# B&R Automation Studio project prak2
Automation Studio 4.5.2.102

## Configuration Config1

### Task classes (Cpu.sw)
```
Cyclic#4:
  Program <- Program.prg
DataObjects: Acp10sys
NcDataObjects: acp10etxen <- acp10etxen.dob
VcDataObjects: LED <- LED.dob
Binaries: udbdef, TCData, vcfntttf, vcpdsw, vcpfmtcx, arial, vcmgr, vccovl, vcdsint, vcpdpp30, vcshared, LED02, LED03, vcpfpp30, LED01, vcalarm, vccbtn, vcptelo, vcgclass, vcdsloc, arialbd, vcrt, vctcal, vcbclass, vcfile, Role, ashwd, ashwac, asfw, iomap, sysconf, User, arconfig, Acp10map, acp10cfg
Libraries: Acp10man, Acp10par, NcGlobal, Acp10sdc, AsBrStr, powerlnk, astime, fileio, runtime, dataobj, vcresman
```

### Hardware
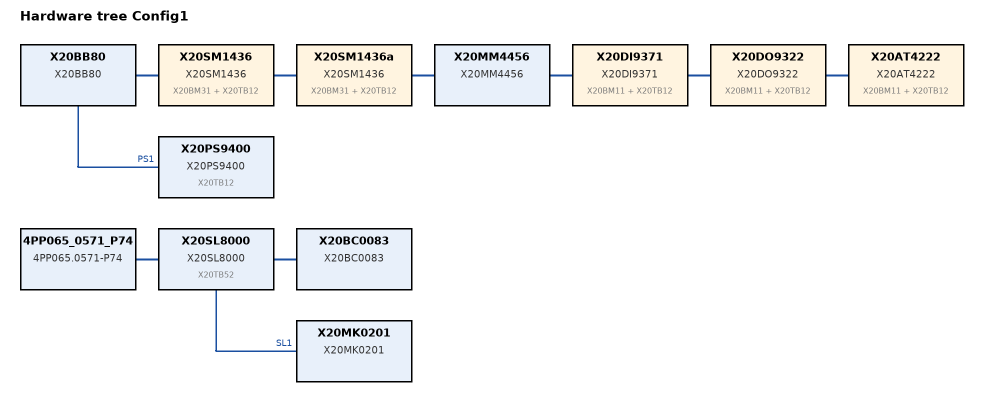
```
4PP065_0571_P74 : 4PP065.0571-P74 v1.1.2.0
  Connector IF5:
    ActivateDevice = 1
    Mode = Manual
    InternetAddress = 10.0.1.10
    SubnetMask = 255.255.255.0
  ConfigurationID = labBR
  TimerDeviceType = EPLX2X
  TimerDevice = 4PP065_0571_P74.IF4
  TaskClassIdleTime = 2000
  Cyclic1Output = 1
  VcObjectName = LED
X20AT4222 : X20AT4222 v1.2.3.0  [SS1 -> X20TB12e.SS; SL -> X20BM11b.SL1]
X20BB80 : X20BB80 v1.0.2.0
X20BC0083 : X20BC0083 v2.14.0.0  [PLK1 -> X20SL8000.PLK2 [Cable Type=PowerlinkCable, Length=10, Version=1.0.0.2]; SL -> X20BB80.SL1]
X20BM11 : X20BM11 v1.0.0.1  [X2X1 -> X20MM4456.X2X2]
X20BM11a : X20BM11 v1.0.0.1  [X2X1 -> X20BM11.X2X2]
X20BM11b : X20BM11 v1.0.0.1  [X2X1 -> X20BM11a.X2X2]
X20BM31 : X20BM31 v1.0.0.1  [X2X1 -> X20BB80.IF1]
X20BM31a : X20BM31 v1.0.0.1  [X2X1 -> X20BM31.X2X2]
X20DI9371 : X20DI9371 v1.0.2.0  [SS1 -> X20TB12c.SS; SL -> X20BM11.SL1]
X20DO9322 : X20DO9322 v1.0.3.0  [SS1 -> X20TB12d.SS; SL -> X20BM11a.SL1]
X20MK0201 : X20MK0201 v1.0.0.0  [SL -> X20SL8000.SL1]
X20MM4456 : X20MM4456 v1.1.5.0  [X2X1 -> X20BM31a.X2X2]
X20PS9400 : X20PS9400 v1.8.0.0  [SS1 -> X20TB12.SS; PS -> X20BB80.PS1]
X20SL8000 : X20SL8000 v1.6.5.2  [PLK1 -> 4PP065_0571_P74.IF4 [Cable Type=PowerlinkCable, Length=10, Version=1.0.0.2]; PLK2 -> X20BC0083.PLK1 [Cable Type=PowerlinkCable, Length=10, Version=1.0.0.2]; SS1 -> X20TB52.SS]
  SafeProject = SafeLOGIC-1
X20SM1436 : X20SM1436 v2.3.0.0  [SS1 -> X20TB12a.SS; SL -> X20BM31.SL1]
  MotionTP = Acp10Arnc0
X20SM1436a : X20SM1436 v2.3.0.0  [SS1 -> X20TB12b.SS; SL -> X20BM31a.SL1]
  MotionTP = Acp10Arnc0
X20TB12 : X20TB12 v1.0.0.0
X20TB12a : X20TB12 v1.0.0.0
X20TB12b : X20TB12 v1.0.0.0
X20TB12c : X20TB12 v1.0.0.0
X20TB12d : X20TB12 v1.0.0.0
X20TB12e : X20TB12 v1.0.0.0
X20TB52 : X20TB52 v1.0.0.1
```

### IoMap.iom - 4PP065_0571_P74/IoMap.iom
```iecst
VAR_CONFIG
	::LED[0] AT %QX."X20DO9322".DigitalOutput02;
	::LED[1] AT %QX."X20DO9322".DigitalOutput03;
	::LED[2] AT %QX."X20DO9322".DigitalOutput04;
	::LED[3] AT %QX."X20DO9322".DigitalOutput05;
END_VAR
```

## Logical view

### Global.var - Global variables
```iecst
VAR
	LED : {REDUND_UNREPLICABLE} ARRAY[0..3] OF BOOL;
END_VAR
```

### Program Logical/Program (ANSIC)

#### Variables.var
```iecst
VAR
	i : INT;
	Button_1 : BOOL;
	Button_2 : BOOL;
	Button_3 : BOOL;
	Button_4 : BOOL;
	press_1 : BOOL;
	press_2 : BOOL;
	press_3 : BOOL;
	press_4 : BOOL;
END_VAR
```

#### Main.c
```c
#include <bur/plctypes.h>

#ifdef _DEFAULT_INCLUDES
	#include <AsDefault.h>
#endif

void _INIT ProgramInit(void)
{
	LED[0] = 0; LED[1] = 1; LED[2] = 0; LED[3] = 1;
	press_1	= 0; press_2	= 0; press_3	= 0; press_4	= 0;
}

void _CYCLIC ProgramCyclic(void)
{
	if(Button_1 && !press_1){
		LED[0] = !LED[0]; LED[1] = !LED[1]; LED[2] = !LED[2];
		press_1 = 1;	}
	if(Button_2 && !press_2){
		LED[0] = !LED[0]; LED[2] = !LED[2];
		press_2 = 1;	}
	if(Button_3 && !press_3){
		LED[1] = !LED[1]; LED[2] = !LED[2]; LED[3] = !LED[3];
		press_3 = 1;	}
	if(Button_4 && !press_4){
		LED[3] = !LED[3];
		press_4 = 1;	}

	if(!Button_1) press_1	= 0;
	if(!Button_2) press_2	= 0;
	if(!Button_3) press_3	= 0;
	if(!Button_4) press_4	= 0;
}

void _EXIT ProgramExit(void)
{

}
```

- Visualisation Logical/LED (not shown)

Listed in the project but not available here: Logical/Global.typ, Logical/Libraries, Logical/acp10etxen
